// TwinCAT 3 PLC project MyPlc
// ProgramVersion: 3.1.4024.0
// libraries:
//   Tc2_SerialCom, * (Beckhoff Automation GmbH)
//   Tc2_Standard, * (Beckhoff Automation GmbH)
//   Tc2_System, * (Beckhoff Automation GmbH)
//   Tc3_Module, * (Beckhoff Automation GmbH)
// project tree:
//   DUTs/ Cylinder.TcPOU, MAX2.TcPOU, TurboPump.TcPOU
//   / PlcTask.TcTTO
//   POUs/ MAIN.TcPOU
// real-time tasks:
//   TASK PlcTask: cycle T#10ms, priority 20, ADS port 350

CONFIGURATION MyPlc
    RESOURCE PLC ON TwinCAT3
        TASK PlcTask(INTERVAL := T#10ms, PRIORITY := 20);
        PROGRAM MAIN WITH PlcTask : MAIN;
    END_RESOURCE
END_CONFIGURATION

// ---- POUs/MAIN.TcPOU
PROGRAM MAIN
VAR
	i : int;
END_VAR

i := i + 1;

END_PROGRAM

// ---- DUTs/Cylinder.TcPOU
// IO元件
FUNCTION_BLOCK PUBLIC Cylinder
VAR_INPUT
END_VAR
VAR_OUTPUT
END_VAR
VAR
END_VAR

END_FUNCTION_BLOCK

// ---- DUTs/MAX2.TcPOU
FUNCTION MAX2 : INT
VAR_INPUT
	a : INT;
	b:INT;
END_VAR
VAR_OUTPUT
	c:INT;
	
END_VAR
VAR
END_VAR

IF a >= b THEN
	MAX2 := a;
	c:=a;
ELSE
	MAX2 := b;
	c:=b;
END_IF

END_FUNCTION

// ---- DUTs/TurboPump.TcPOU
// SerialPort元件
FUNCTION_BLOCK TurboPump
VAR_INPUT
	SetTmsTemp_CmdTransId:UINT;
END_VAR
VAR_OUTPUT
	SetTmsTemp_EchoTransId : UINT;
	SetTmsTemp_ErrorCode:BYTE;
END_VAR
VAR
	
END_VAR

IF SetTmsTemp_CmdTransId <> SetTmsTemp_EchoTransId THEN
	IF SetTmsTemp_ErrorCode <> 0 THEN
		SetTmsTemp(temp:= 100);
		SetTmsTemp_ErrorCode := 1;
	END_IF
END_IF

METHOD PUBLIC SetTmsTemp
VAR_INPUT
	temp :REAL;
END_VAR
END_METHOD

END_FUNCTION_BLOCK
